// TIA Portal V19 export
FUNCTION "EXCHANGETRAY_CallMaterials" : Void   // FC3, LAD
// stored: SetENOAutomatically false
BEGIN

REGION Network 1: U1 Constraint
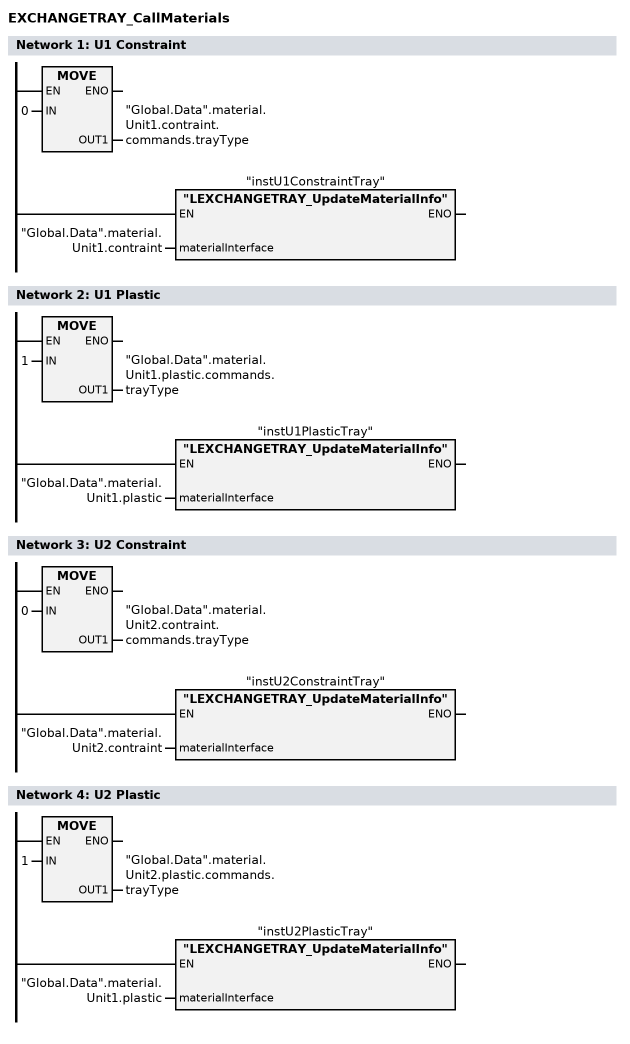
   RUNG wire#powerrail
      Move(in := 0, out1 => "Global.Data".material.Unit1.contraint.commands.trayType)
   END_RUNG
   RUNG wire#powerrail
      "instU1ConstraintTray"(materialInterface := "Global.Data".material.Unit1.contraint)
   END_RUNG
   // the same network as SCL:
   "Global.Data".material.Unit1.contraint.commands.trayType := 0;
   "instU1ConstraintTray"(materialInterface := "Global.Data".material.Unit1.contraint);   // "LEXCHANGETRAY_UpdateMaterialInfo"
END_REGION

REGION Network 2: U1 Plastic
   RUNG wire#powerrail
      Move(in := 1, out1 => "Global.Data".material.Unit1.plastic.commands.trayType)
   END_RUNG
   RUNG wire#powerrail
      "instU1PlasticTray"(materialInterface := "Global.Data".material.Unit1.plastic)
   END_RUNG
   // the same network as SCL:
   "Global.Data".material.Unit1.plastic.commands.trayType := 1;
   "instU1PlasticTray"(materialInterface := "Global.Data".material.Unit1.plastic);   // "LEXCHANGETRAY_UpdateMaterialInfo"
END_REGION

REGION Network 3: U2 Constraint
   RUNG wire#powerrail
      Move(in := 0, out1 => "Global.Data".material.Unit2.contraint.commands.trayType)
   END_RUNG
   RUNG wire#powerrail
      "instU2ConstraintTray"(materialInterface := "Global.Data".material.Unit2.contraint)
   END_RUNG
   // the same network as SCL:
   "Global.Data".material.Unit2.contraint.commands.trayType := 0;
   "instU2ConstraintTray"(materialInterface := "Global.Data".material.Unit2.contraint);   // "LEXCHANGETRAY_UpdateMaterialInfo"
END_REGION

REGION Network 4: U2 Plastic
   RUNG wire#powerrail
      Move(in := 1, out1 => "Global.Data".material.Unit2.plastic.commands.trayType)
   END_RUNG
   RUNG wire#powerrail
      "instU2PlasticTray"(materialInterface := "Global.Data".material.Unit1.plastic)
   END_RUNG
   // the same network as SCL:
   "Global.Data".material.Unit2.plastic.commands.trayType := 1;
   "instU2PlasticTray"(materialInterface := "Global.Data".material.Unit1.plastic);   // "LEXCHANGETRAY_UpdateMaterialInfo"
END_REGION
END_FUNCTION
